TYPE ST_SlaveDynaData :
STRUCT
	// mass matrix in joint space
	m_massMat :ARRAY[1..g_sArmNum] OF Mat3d;
	
	// gravity
	m_gravity :ARRAY[1..g_sArmNum] OF Vec3d;
	
	// instrument out-of-view data
	m_insruViewData :ARRAY[1..g_sArmNum] OF Vec3i;
END_STRUCT
END_TYPE

(* stored: Version 1.1.0.1, ProductVersion 3.1.4024.12
   DUT ST_SlaveDynaData: Id {720ec479-04e0-4039-9c54-19b1d24e2b5b} *)
